// TIA Portal V18 export
// export: Created 2026-06-11T19:03:46.1512647Z, ExportSetting WithDefaults, DisplayName Totally Integrated Automation Portal, DisplayVersion V18, DisplayName TIA Portal Openness, DisplayVersion V18, DisplayName TIA Portal Version Control Interface, DisplayVersion V18, DisplayName STEP 7 Professional, DisplayVersion V18, DisplayName STEP 7 Safety, DisplayVersion V18, DisplayName WinCC Professional, DisplayVersion V18
Screen "scadabai5"  1920x1080, Number=6
  ScreenLayer 
    GraphicView "Graphic view_1" at 0,0 size 1920x1080  Picture=anh nen
    Circle "Circle_1" at 8,51 size 19x19
    Circle "Circle_2" at 8,68 size 19x19
    Circle "Circle_3" at 8,87 size 19x19
    Circle "Circle_4" at 180,52 size 19x19
    Circle "Circle_5" at 181,70 size 19x19
    Circle "Circle_6" at 250,175 size 19x19
    Circle "Circle_7" at 122,242 size 18x18
    Circle "Circle_8" at 122,259 size 18x18
    Circle "Circle_9" at 122,277 size 19x19
    Circle "Circle_10" at 86,316 size 19x19
    Circle "Circle_11" at 188,316 size 19x19
    Circle "Circle_12" at 283,316 size 19x19
    GraphicView "Graphic view_2" at 194,49 size 90x150  Picture=bon
    Circle "Circle_13" at 217,166 size 32x32
    Circle "Circle_14" at 39,392 size 19x19
    Circle "Circle_15" at 144,392 size 17x17
    Circle "Circle_16" at 238,391 size 17x17
    Button "Button_5" at 1704,197 size 39x37  Mode=Text, TextOn="Text"
    Button "Button_6" at 1740,45 size 171x35  Mode=Text, TextOff="TRANSPORT GROUP", TextOn="Text"
    Button "Button_7" at 1742,85 size 171x35  Mode=Text, TextOff="GAS FLOW GROUP", TextOn="Text"
    Button "Button_8" at 1741,116 size 172x37  Mode=Text, TextOff="LUB GROUP", TextOn="Text"
    Button "Button_9" at 1742,154 size 170x36  Mode=Text, TextOff="CEMENT MILL GROUP", TextOn="Text"
    Button "Button_10" at 1742,198 size 171x35  Mode=Text, TextOff="CM FEED GROUP", TextOn="Text"
    Button "Button_11" at 1698,242 size 220x24  Mode=Text, TextOff="ALARM RESET", TextOn="Text"
    Button "Button_12" at 1698,268 size 220x22  Mode=Text, TextOff="CM DAMFERS", TextOn="Text"
    Button "Button_13" at 1698,293 size 220x34  Mode=Text, TextOff="INTERLOCKS", TextOn="Text"
    TextField "Text field_1" at 228,171 size 12x19  Text="M"
    Circle "Circle_17" at 86,152 size 30x30
    Circle "Circle_18" at 118,152 size 30x30
    Circle "Circle_19" at 73,77 size 33x33
    TextField "Text field_2" at 95,158 size 12x19  Text="M"
    TextField "Text field_3" at 129,157 size 12x19  Text="M"
    TextField "Text field_4" at 83,83 size 12x19  Text="M"
    Circle "Circle_20" at 257,257 size 30x30
    TextField "Text field_5" at 267,264 size 12x19  Text="M"
    IOField "I/O field_1" at 53,455 size 57x22  DataFormat=Decimal, FormatPattern=99.9, Mode=InOutput
      ProcessValue := AI_B5_CA_Fan_Motor_DE_Temp
    IOField "I/O field_2" at 54,485 size 54x22  DataFormat=Decimal, FormatPattern=99.9, Mode=InOutput
      ProcessValue := AI_B5_CA_Fan_Motor_NDE_Temp
    IOField "I/O field_3" at 54,515 size 55x22  DataFormat=Decimal, FormatPattern=99.9, Mode=InOutput
      ProcessValue := AI_B5_CA_Fan_DE_Temp
    IOField "I/O field_4" at 157,455 size 55x22  DataFormat=Decimal, FormatPattern=99.9, Mode=InOutput
      ProcessValue := AI_B5_CA_Fan_NDE_Temp
    IOField "I/O field_5" at 156,488 size 56x22  DataFormat=Decimal, FormatPattern=99.9, Mode=InOutput
      ProcessValue := AI_B5_CA_Fan_DE_Vib
    IOField "I/O field_6" at 155,516 size 58x24  DataFormat=Decimal, FormatPattern=99.9, Mode=InOutput
      ProcessValue := AI_B5_CA_Fan_NDE_Vib
    IOField "I/O field_7" at 259,453 size 53x24  DataFormat=Decimal, FormatPattern=999.9, Mode=InOutput
      ProcessValue := AI_B5_SP_700FN03
    IOField "I/O field_8" at 259,483 size 54x22  DataFormat=Decimal, FormatPattern=999.9, Mode=InOutput
      ProcessValue := AI_B5_SP_700HES01
    IOField "I/O field_9" at 259,512 size 54x23  DataFormat=Decimal, FormatPattern=99.9, Mode=InOutput
      ProcessValue := AI_B5_SP_700DA4
    IOField "I/O field_10" at 482,376 size 59x17  DataFormat=Decimal, FormatPattern=99.9, Mode=InOutput
      ProcessValue := AI_B5_SP_700DA6
    IOField "I/O field_11" at 482,396 size 59x17  DataFormat=Decimal, FormatPattern=99.9, Mode=InOutput
      ProcessValue := AI_B5_SP_700DA7
    IOField "I/O field_12" at 482,416 size 59x18  DataFormat=Decimal, FormatPattern=99.9, Mode=InOutput
      ProcessValue := AI_B5_SP_700FN2_DA1
    IOField "I/O field_13" at 481,435 size 59x17  DataFormat=Decimal, FormatPattern=99.9, Mode=InOutput
      ProcessValue := AI_B5_Sep_Motor_Top_Temp
    IOField "I/O field_14" at 481,455 size 59x17  DataFormat=Decimal, FormatPattern=99.9, Mode=InOutput
      ProcessValue := AI_B5_Sep_Bottom_Bear_Temp
    IOField "I/O field_15" at 481,476 size 59x17  DataFormat=Decimal, FormatPattern=999.9, Mode=InOutput
      ProcessValue := AI_B5_Trend_Val_1
    IOField "I/O field_16" at 482,513 size 57x17  DataFormat=Decimal, FormatPattern=999.9, Mode=InOutput
      ProcessValue := AI_B5_Trend_Val_2
    IOField "I/O field_17" at 482,536 size 58x18  DataFormat=Decimal, FormatPattern=999.9, Mode=InOutput
      ProcessValue := AI_B5_Trend_Val_3
    IOField "I/O field_18" at 647,377 size 59x17  DataFormat=Decimal, FormatPattern=999.9, Mode=InOutput
      ProcessValue := AI_B5_700FN03_RPM
    IOField "I/O field_19" at 646,397 size 59x18  DataFormat=Decimal, FormatPattern=999.9, Mode=InOutput
      ProcessValue := AI_B5_700HES01_Flow
    IOField "I/O field_20" at 647,414 size 59x17  DataFormat=Decimal, FormatPattern=99.9, Mode=InOutput
      ProcessValue := AI_B5_700FN10_Speed
    IOField "I/O field_21" at 647,436 size 59x17  DataFormat=Decimal, FormatPattern=999.9, Mode=InOutput
      ProcessValue := AI_B5_700CM01_Current
    IOField "I/O field_22" at 647,457 size 59x17  DataFormat=Decimal, FormatPattern=999.9, Mode=InOutput
      ProcessValue := AI_B5_Lub_Stop_Time
    IOField "I/O field_23" at 647,479 size 58x17  DataFormat=Decimal, FormatPattern=999.9, Mode=InOutput
      ProcessValue := AI_B5_Main_Drive_ReHealth
    IOField "I/O field_24" at 334,648 size 58x23  DataFormat=Decimal, FormatPattern=99.9, Mode=InOutput
      ProcessValue := AI_B5_CM_LRS_IN
    IOField "I/O field_25" at 334,674 size 58x22  DataFormat=Decimal, FormatPattern=99.9, Mode=InOutput
      ProcessValue := AI_B5_CM_LRS_OUT
    IOField "I/O field_26" at 156,583 size 54x23  DataFormat=Decimal, FormatPattern=99.9, Mode=InOutput
      ProcessValue := AI_B5_CM_Mill_Oil_Temp
    IOField "I/O field_27" at 252,584 size 53x22  DataFormat=Decimal, FormatPattern=99.9, Mode=InOutput
      ProcessValue := AI_B5_CM_OilTrun_BER_Temp
    IOField "I/O field_28" at 765,382 size 59x22  DataFormat=Decimal, FormatPattern=99.9, Mode=InOutput
      ProcessValue := AI_B5_CM_OilTrun_BER2_Temp
    IOField "I/O field_29" at 876,299 size 57x26  DataFormat=Decimal, FormatPattern=99.9, Mode=InOutput
      ProcessValue := AI_B5_CM_OilPinion_BER_Temp
    IOField "I/O field_30" at 925,369 size 57x24  DataFormat=Decimal, FormatPattern=99.9, Mode=InOutput
      ProcessValue := AI_B5_CM_GB_IL_Shaft_BER
    IOField "I/O field_31" at 924,400 size 59x22  DataFormat=Decimal, FormatPattern=999.9, Mode=InOutput
      ProcessValue := AI_B5_CM_Running_Hours
    IOField "I/O field_32" at 824,88 size 59x23  DataFormat=Decimal, FormatPattern=99.9, Mode=InOutput
      ProcessValue := AI_B5_CM_PS1_1_KG
    IOField "I/O field_33" at 1062,42 size 56x23  DataFormat=Decimal, FormatPattern=99.9, Mode=InOutput
      ProcessValue := AI_B5_CM_PS1_2_KG
    IOField "I/O field_34" at 1375,249 size 56x21  DataFormat=Decimal, FormatPattern=999.9, Mode=InOutput
      ProcessValue := AI_B5_NIBS_Value
    IOField "I/O field_40" at 500,885 size 55x18  DataFormat=Decimal, FormatPattern=999.9, Mode=InOutput
      ProcessValue := AI_B5_800YF2_Flow
    IOField "I/O field_41" at 501,904 size 52x16  DataFormat=Decimal, FormatPattern=999.9, Mode=InOutput
      ProcessValue := AI_B5_Silo1_Level_Bar1
    IOField "I/O field_42" at 626,631 size 58x22  DataFormat=Decimal, FormatPattern=999.9, Mode=InOutput
      ProcessValue := AI_B5_Silo1_Level_Bar2
    IOField "I/O field_43" at 641,714 size 58x22  DataFormat=Decimal, FormatPattern=999.9, Mode=InOutput
      ProcessValue := AI_B5_Silo2_Level_Bar1
    IOField "I/O field_44" at 690,812 size 59x22  DataFormat=Decimal, FormatPattern=999.9, Mode=InOutput
      ProcessValue := AI_B5_Silo2_Level_Bar2
    IOField "I/O field_45" at 757,909 size 58x22  DataFormat=Decimal, FormatPattern=99.9, Mode=InOutput
      ProcessValue := AI_B5_700FN01_Speed
    IOField "I/O field_46" at 878,891 size 52x22  DataFormat=Decimal, FormatPattern=99.9, Mode=InOutput
      ProcessValue := AI_B5_700FN02_Speed
    IOField "I/O field_47" at 954,696 size 58x22  DataFormat=Decimal, FormatPattern=99.9, Mode=InOutput
      ProcessValue := AI_B5_700AS07_Speed
    IOField "I/O field_48" at 1062,835 size 51x22  DataFormat=Decimal, FormatPattern=999.9, Mode=InOutput
      ProcessValue := AI_B5_700AS08_Flow
    IOField "I/O field_49" at 1137,789 size 58x22  DataFormat=Decimal, FormatPattern=99.9, Mode=InOutput
      ProcessValue := AI_B5_700FN09_Speed
    IOField "I/O field_50" at 1131,949 size 58x22  DataFormat=Decimal, FormatPattern=99.9, Mode=InOutput
      ProcessValue := AI_B5_700SFM01_Speed
    IOField "I/O field_51" at 1381,929 size 58x21  DataFormat=Decimal, FormatPattern=999.9, Mode=InOutput
      ProcessValue := AI_B5_700DA1_Flow
    IOField "I/O field_52" at 1391,790 size 58x21  DataFormat=Decimal, FormatPattern=999.9, Mode=InOutput
      ProcessValue := AI_B5_700DA4_Flow
    IOField "I/O field_53" at 1768,859 size 58x24  DataFormat=Decimal, FormatPattern=99.9, Mode=InOutput
      ProcessValue := AI_B5_700DA6_Temp
    IOField "I/O field_54" at 465,956 size 49x16  DataFormat=Decimal, FormatPattern=99.9, Mode=InOutput
      ProcessValue := AI_B5_700DA7_Temp
    IOField "I/O field_55" at 523,957 size 49x16  DataFormat=Decimal, FormatPattern=999.9, Mode=InOutput
      ProcessValue := AI_B5_700BL1_Load
    IOField "I/O field_56" at 246,862 size 58x23  DataFormat=Decimal, FormatPattern=999.9, Mode=InOutput
      ProcessValue := AI_B5_700BL2_Load
    Circle "Circle_21" at 286,82 size 32x32
    TextField "Text field_6" at 296,88 size 12x19  Text="M"
    Circle "Circle_22" at 86,416 size 30x30
    Circle "Circle_23" at 192,416 size 28x28
    Circle "Circle_24" at 288,414 size 31x31
    Circle "Circle_25" at 98,612 size 18x18
    Circle "Circle_26" at 162,612 size 18x18
    Circle "Circle_27" at 226,613 size 18x18
    Circle "Circle_28" at 74,705 size 25x25
    TextField "Text field_7" at 94,423 size 12x19  Text="M"
    TextField "Text field_8" at 201,421 size 12x19  Text="M"
    TextField "Text field_9" at 299,421 size 12x19  Text="M"
    TextField "Text field_10" at 81,708 size 12x19  Text="M"
    Circle "Circle_29" at 138,706 size 25x25
    Circle "Circle_30" at 177,706 size 25x25
    Circle "Circle_31" at 177,772 size 25x25
    Circle "Circle_32" at 138,772 size 25x25
    Circle "Circle_33" at 73,772 size 25x25
    TextField "Text field_11" at 144,709 size 12x19  Text="M"
    TextField "Text field_12" at 184,709 size 12x19  Text="M"
    TextField "Text field_13" at 184,774 size 12x19  Text="M"
    TextField "Text field_14" at 145,775 size 12x19  Text="M"
    TextField "Text field_15" at 80,776 size 12x19  Text="M"
    Circle "Circle_34" at 74,846 size 25x25
    Circle "Circle_35" at 138,845 size 25x25
    Circle "Circle_36" at 73,916 size 25x25
    Circle "Circle_37" at 142,916 size 17x17
    Circle "Circle_38" at 176,915 size 17x17
    Circle "Circle_39" at 210,915 size 17x17
    Circle "Circle_40" at 243,916 size 17x17
    Circle "Circle_41" at 141,950 size 17x17
    TextField "Text field_16" at 81,848 size 12x19  Text="M"
    TextField "Text field_17" at 144,848 size 12x19  Text="M"
    Circle "Circle_42" at 408,727 size 17x17
    Circle "Circle_43" at 407,746 size 17x17
    Circle "Circle_44" at 408,764 size 17x17
    Bar "Bar_1" at 1622,837 size 85x126  CountSubDivisions=2, IntegerDigits=2, LargeTickLabelingStep=1, MaximumValue=25, Precision=2
    Bar "Bar_2" at 1914,794 size 86x124  CountSubDivisions=2, IntegerDigits=2, LargeTickLabelingStep=1, MaximumValue=25, Precision=2
    IOField "I/O field_57" at 945,188 size 59x21  DataFormat=Decimal, FormatPattern=999.9, Mode=InOutput
      ProcessValue := AI_B5_700AS9_Flow
    IOField "I/O field_58" at 946,213 size 58x23  DataFormat=Decimal, FormatPattern=99.9, Mode=InOutput
      ProcessValue := AI_B5_700FN13_Speed
    Button "Button_14" at 98,190 size 39x23  Mode=Text, TextOff="Text", TextOn="Text"
    Button "Button_15" at 18,454 size 33x24  Mode=Text, TextOff="Text", TextOn="Text"
    Button "Button_16" at 18,485 size 33x24  Mode=Text, TextOff="Text", TextOn="Text"
    Button "Button_17" at 119,454 size 34x23  Mode=Text, TextOff="Text", TextOn="Text"
    Button "Button_18" at 119,486 size 33x23  Mode=Text, TextOff="Text", TextOn="Text"
    Button "Button_19" at 223,486 size 33x23  Mode=Text, TextOff="Text", TextOn="Text"
    Button "Button_20" at 223,455 size 33x23  Mode=Text, TextOff="Text", TextOn="Text"
    Button "Button_21" at 249,950 size 66x33  Mode=Text, TextOff="LOS", TextOn="Text"
    Button "Button_22" at 11,711 size 60x49  Mode=Text, TextOff="LQ 61", TextOn="Text"
    Button "Button_23" at 13,775 size 58x46  Mode=Text, TextOff="LQ 62", TextOn="Text"
    Button "Button_24" at 13,836 size 57x49  Mode=Text, TextOff="ELS", TextOn="Text"
    Button "Button_25" at 13,922 size 58x55  Mode=Text, TextOff="LQ 63", TextOn="Text"
    Circle "Circle_45" at 560,578 size 33x33
    TextField "Text field_18" at 570,585 size 12x19  Text="M"
    Circle "Circle_46" at 796,584 size 32x32
    Circle "Circle_47" at 868,585 size 29x29
    TextField "Text field_19" at 805,589 size 12x19  Text="M"
    TextField "Text field_20" at 878,590 size 12x19  Text="M"
    Circle "Circle_48" at 772,764 size 33x33
    TextField "Text field_21" at 784,772 size 12x19  Text="M"
    Circle "Circle_49" at 769,860 size 33x33
    TextField "Text field_22" at 779,867 size 12x19  Text="M"
    Circle "Circle_50" at 740,855 size 22x22
    TextField "Text field_23" at 745,856 size 12x19  Text="M"
    Circle "Circle_51" at 898,860 size 22x22
    TextField "Text field_24" at 903,861 size 12x19  Text="M"
    Circle "Circle_52" at 895,947 size 14x14
    Circle "Circle_53" at 895,961 size 14x14
    Circle "Circle_54" at 970,921 size 31x31
    TextField "Text field_25" at 980,926 size 12x19  Text="M"
    Circle "Circle_55" at 1014,921 size 31x31
    TextField "Text field_26" at 1024,928 size 12x19  Text="M"
    Circle "Circle_56" at 808,464 size 19x19
    Circle "Circle_57" at 833,460 size 25x25
    Circle "Circle_58" at 877,461 size 25x25
    Circle "Circle_59" at 908,464 size 19x19
    Circle "Circle_60" at 985,464 size 19x19
    Circle "Circle_61" at 1009,458 size 25x25
    Circle "Circle_62" at 1289,433 size 33x33
    Circle "Circle_63" at 1086,464 size 19x19
    TextField "Text field_27" at 839,464 size 12x19  Text="M"
    TextField "Text field_28" at 883,464 size 12x19  Text="M"
    TextField "Text field_30" at 1299,440 size 12x19  Text="M"
    Circle "Circle_64" at 934,314 size 41x41
    TextField "Text field_31" at 948,326 size 12x19  Text="M"
    Circle "Circle_65" at 958,115 size 33x33
    TextField "Text field_32" at 968,120 size 12x19  Text="M"
    Circle "Circle_66" at 1100,209 size 30x30
    TextField "Text field_33" at 1110,213 size 12x19  Text="M"
    Circle "Circle_67" at 1147,62 size 33x33
    TextField "Text field_34" at 1156,68 size 12x19  Text="M"
    Circle "Circle_68" at 1188,95 size 18x18
    Circle "Circle_69" at 1316,52 size 19x19
    Circle "Circle_70" at 1317,70 size 19x19
    Circle "Circle_71" at 1335,166 size 19x19
    Circle "Circle_72" at 1357,79 size 31x31
    Circle "Circle_73" at 1357,157 size 30x30
    Circle "Circle_74" at 1459,135 size 30x30
    Circle "Circle_75" at 1454,218 size 30x30
    Circle "Circle_76" at 1298,282 size 30x30
    TextField "Text field_35" at 1308,287 size 12x19  Text="M"
    TextField "Text field_36" at 1368,85 size 12x19  Text="M"
    TextField "Text field_37" at 1430,152 size 12x19  Text="M"
    TextField "Text field_38" at 1367,164 size 12x19  Text="M"
    TextField "Text field_39" at 1463,224 size 12x19  Text="M"
    Circle "Circle_77" at 1155,920 size 22x22
    Circle "Circle_78" at 1236,385 size 19x19
    Circle "Circle_79" at 1236,406 size 19x19
    Circle "Circle_80" at 1379,495 size 19x19
    Circle "Circle_81" at 1489,372 size 19x19
    Circle "Circle_82" at 1489,391 size 19x19
    Circle "Circle_83" at 1272,530 size 19x19
    Circle "Circle_84" at 1401,488 size 36x36
    TextField "Text field_40" at 1413,496 size 12x19  Text="M"
    Circle "Circle_85" at 1526,479 size 36x36
    TextField "Text field_41" at 1536,488 size 12x19  Text="M"
    Circle "Circle_86" at 1603,397 size 31x31
    TextField "Text field_42" at 1614,404 size 12x19  Text="M"
    Circle "Circle_87" at 1532,399 size 31x31
    TextField "Text field_43" at 1542,405 size 12x19  Text="M"
    Circle "Circle_88" at 1713,481 size 31x31
    TextField "Text field_44" at 1722,488 size 12x19  Text="M"
    Circle "Circle_89" at 1564,490 size 19x19
    Circle "Circle_90" at 1672,373 size 19x19
    Circle "Circle_91" at 1673,393 size 19x19
    Circle "Circle_92" at 1693,488 size 19x19
    Circle "Circle_93" at 1788,399 size 31x31
    Circle "Circle_94" at 1792,458 size 31x31
    Circle "Circle_95" at 1712,394 size 31x31
    TextField "Text field_45" at 1797,406 size 12x19  Text="M"
    TextField "Text field_46" at 1722,400 size 12x19  Text="M"
    TextField "Text field_47" at 1801,465 size 12x19  Text="M"
    Circle "Circle_96" at 1580,600 size 31x31
    TextField "Text field_48" at 1590,608 size 12x19  Text="M"
    Circle "Circle_97" at 1473,769 size 31x31
    TextField "Text field_49" at 1483,774 size 12x19  Text="M"
    Circle "Circle_98" at 1301,889 size 31x31
    TextField "Text field_50" at 1311,894 size 12x19  Text="M"
    Circle "Circle_99" at 1234,888 size 31x31
    TextField "Text field_51" at 1244,894 size 12x19  Text="M"
    Circle "Circle_100" at 1411,885 size 17x17
    Circle "Circle_101" at 1687,769 size 31x31
    TextField "Text field_52" at 1696,774 size 12x19  Text="M"
    Button "Button_26" at 1529,929 size 78x23  Mode=Text, TextOff="SELECTED", TextOn="Text"
    Circle "Circle_102" at 1506,840 size 20x20
    Circle "Circle_103" at 1723,842 size 20x20
    Button "Button_28" at 179,1024 size 173x20  Mode=Text, TextOff="REPORT", TextOn="Text"
    Button "Button_29" at 178,1049 size 172x24  Mode=Text, TextOff="TRENDS", TextOn="Text"
    Button "Button_30" at 357,1024 size 167x20  Mode=Text, TextOff="RAW MILL", TextOn="Text"
    Button "Button_31" at 355,1048 size 168x25  Mode=Text, TextOff="ALARM", TextOn="Text"
    Button "Button_32" at 527,1021 size 171x23  Mode=Text, TextOff="BLENDING SILO", TextOn="Text"
    Button "Button_33" at 527,1049 size 172x23  Mode=Text, TextOff="FLYASH SILO", TextOn="Text"
    Button "Button_34" at 700,1021 size 172x25  Mode=Text, TextOff="COAL MILL", TextOn="Text"
    Button "Button_35" at 700,1047 size 173x25  Mode=Text, TextOff="INSTRUCTIONS", TextOn="Text"
    Button "Button_36" at 875,1021 size 169x25  Mode=Text, TextOff="GREATE COOLER", TextOn="Text"
    Button "Button_37" at 1047,1018 size 171x25  Mode=Text, TextOff="KILN GROUP", TextOn="Text"
    Button "Button_38" at 1220,1020 size 175x25  Mode=Text, TextOff="HOPPER FEEDING", TextOn="Text"
    Button "Button_39" at 1398,1018 size 169x25  Mode=Text, TextOff="CEM MILL GROUP", TextOn="Text"
    Button "Button_40" at 1566,1019 size 180x25  Mode=Text, TextOff="EXTR.& PACKING", TextOn="Text"
    Button "Button_41" at 874,1047 size 172x25  Mode=Text, TextOff="RUNNING HOURS", TextOn="Text"
    Button "Button_42" at 1047,1047 size 171x25  Mode=Text, TextOff="SPARE", TextOn="Text"
    Button "Button_43" at 1222,1047 size 170x25  Mode=Text, TextOff="HOOTER", TextOn="Text"
    Button "Button_44" at 1396,1048 size 169x25  Mode=Text, TextOff="EXIT", TextOn="Text"
    Button "Button_45" at 1565,1048 size 180x25  Mode=Text, TextOff="ABOUT", TextOn="Text"
    IOField "I/O field_35" at 500,865 size 55x18  DataFormat=Decimal, FormatPattern=99.9, Mode=InOutput
      ProcessValue := AI_B5_800DC1_Temp
    IOField "I/O field_36" at 500,845 size 55x18  DataFormat=Decimal, FormatPattern=99.9, Mode=InOutput
      ProcessValue := AI_B5_800DC2_Temp
    Bar "Bar_3" at 1822,834 size 85x126  CountSubDivisions=2, IntegerDigits=2, LargeTickLabelingStep=1, MaximumValue=25, Precision=2
    IOField "I/O field_37" at 500,825 size 55x18  DataFormat=Decimal, FormatPattern=99.9, Mode=InOutput
      ProcessValue := AI_B5_800FN1_Speed
    IOField "I/O field_38" at 500,805 size 55x18  DataFormat=Decimal, FormatPattern=99.9, Mode=InOutput
      ProcessValue := AI_B5_800FN2_Speed
    IOField "I/O field_39" at 500,785 size 55x18  DataFormat=Decimal, FormatPattern=999.9, Mode=InOutput
      ProcessValue := AI_B5_800YF1_Flow
    Button "Button_27" at 1756,929 size 78x23  Mode=Text, TextOff="SELECTED", TextOn="Text"
    Button "Button_1" at 1704,159 size 39x37  Mode=Text, TextOn="Text"
    Button "Button_2" at 1704,121 size 39x37  Mode=Text, TextOn="Text"
    Button "Button_3" at 1704,83 size 39x37  Mode=Text, TextOn="Text"
    Button "Button_4" at 1704,45 size 39x37  Mode=Text, TextOn="Text"
    Circle "Circle_104" at 1292,522 size 33x33
    TextField "Text field_29" at 1304,530 size 12x19  Text="M"
    Circle "Circle_105" at 1055,460 size 24x24
    TextField "Text field_53" at 1061,463 size 12x19  Text="M"
    TextField "Text field_54" at 1015,462 size 12x19  Text="M"
    Circle "Circle_106" at 1082,587 size 29x29
    TextField "Text field_55" at 1090,594 size 12x19  Text="M"
    Button "Btn_Enter_System_4" at 1806,0 size 114x38  Mode=Text, StyleItem=Button, TextOff="Mh login", TextOn="Text"
      VisibilityAnimation "VisibilityAnimation"  RangeEnd=99, RangeStart=1
        tag Logged_In
      on Click: ActivateScreen(Screen name := Login/out, Object number := 0)
    TextField "Text_field_Unit_I/O field_1" at 118,455 size 50x22  Text="<body><p>°C</p></body>"
    TextField "Text_field_Unit_I/O field_2" at 116,485 size 50x22  Text="<body><p>°C</p></body>"
    TextField "Text_field_Unit_I/O field_3" at 117,515 size 50x22  Text="<body><p>°C</p></body>"
    TextField "Text_field_Unit_I/O field_4" at 220,455 size 50x22  Text="<body><p>°C</p></body>"
    TextField "Text_field_Unit_I/O field_5" at 220,488 size 50x22  Text="<body><p>mm/s</p></body>"
    TextField "Text_field_Unit_I/O field_6" at 221,516 size 50x24  Text="<body><p>mm/s</p></body>"
    TextField "Text_field_Unit_I/O field_7" at 320,453 size 50x24  Text="<body><p>L/h</p></body>"
    TextField "Text_field_Unit_I/O field_8" at 321,483 size 50x22  Text="<body><p>L/h</p></body>"
    TextField "Text_field_Unit_I/O field_9" at 321,512 size 50x23  Text="<body><p>Hz</p></body>"
    TextField "Text_field_Unit_I/O field_10" at 549,376 size 50x17  Text="<body><p>Hz</p></body>"
    TextField "Text_field_Unit_I/O field_11" at 549,396 size 50x17  Text="<body><p>Hz</p></body>"
    TextField "Text_field_Unit_I/O field_12" at 549,416 size 50x18  Text="<body><p>Hz</p></body>"
    TextField "Text_field_Unit_I/O field_13" at 548,435 size 50x17  Text="<body><p>°C</p></body>"
    TextField "Text_field_Unit_I/O field_14" at 548,455 size 50x17  Text="<body><p>°C</p></body>"
    TextField "Text_field_Unit_I/O field_15" at 548,476 size 50x17  Text="<body><p>%</p></body>"
    TextField "Text_field_Unit_I/O field_16" at 547,513 size 50x17  Text="<body><p>%</p></body>"
    TextField "Text_field_Unit_I/O field_17" at 548,536 size 50x18  Text="<body><p>%</p></body>"
    TextField "Text_field_Unit_I/O field_18" at 714,377 size 50x17  Text="<body><p>RPM</p></body>"
    TextField "Text_field_Unit_I/O field_19" at 713,397 size 50x18  Text="<body><p>L/h</p></body>"
    TextField "Text_field_Unit_I/O field_20" at 714,414 size 50x17  Text="<body><p>Hz</p></body>"
    TextField "Text_field_Unit_I/O field_21" at 714,436 size 50x17  Text="<body><p>A</p></body>"
    TextField "Text_field_Unit_I/O field_22" at 714,457 size 50x17  Text="<body><p>Sec</p></body>"
    TextField "Text_field_Unit_I/O field_23" at 713,479 size 50x17  Text="<body><p>Sec</p></body>"
    TextField "Text_field_Unit_I/O field_24" at 400,648 size 50x23  Text="<body><p>°C</p></body>"
    TextField "Text_field_Unit_I/O field_25" at 400,674 size 50x22  Text="<body><p>°C</p></body>"
    TextField "Text_field_Unit_I/O field_26" at 218,583 size 50x23  Text="<body><p>°C</p></body>"
    TextField "Text_field_Unit_I/O field_27" at 313,584 size 50x22  Text="<body><p>°C</p></body>"
    TextField "Text_field_Unit_I/O field_28" at 832,382 size 50x22  Text="<body><p>°C</p></body>"
    TextField "Text_field_Unit_I/O field_29" at 941,299 size 50x26  Text="<body><p>°C</p></body>"
    TextField "Text_field_Unit_I/O field_30" at 990,369 size 50x24  Text="<body><p>°C</p></body>"
    TextField "Text_field_Unit_I/O field_31" at 991,400 size 50x22  Text="<body><p>Hr</p></body>"
    TextField "Text_field_Unit_I/O field_32" at 891,88 size 50x23  Text="<body><p>bar</p></body>"
    TextField "Text_field_Unit_I/O field_33" at 1126,42 size 50x23  Text="<body><p>bar</p></body>"
    TextField "Text_field_Unit_I/O field_34" at 1439,249 size 50x21  Text="<body><p>A</p></body>"
    TextField "Text_field_Unit_I/O field_40" at 563,885 size 50x18  Text="<body><p>L/h</p></body>"
    TextField "Text_field_Unit_I/O field_41" at 561,904 size 50x16  Text="<body><p>%</p></body>"
    TextField "Text_field_Unit_I/O field_42" at 692,631 size 50x22  Text="<body><p>%</p></body>"
    TextField "Text_field_Unit_I/O field_43" at 707,714 size 50x22  Text="<body><p>%</p></body>"
    TextField "Text_field_Unit_I/O field_44" at 757,812 size 50x22  Text="<body><p>%</p></body>"
    TextField "Text_field_Unit_I/O field_45" at 823,909 size 50x22  Text="<body><p>Hz</p></body>"
    TextField "Text_field_Unit_I/O field_46" at 938,891 size 50x22  Text="<body><p>Hz</p></body>"
    TextField "Text_field_Unit_I/O field_47" at 1020,696 size 50x22  Text="<body><p>Hz</p></body>"
    TextField "Text_field_Unit_I/O field_48" at 1121,835 size 50x22  Text="<body><p>L/h</p></body>"
    TextField "Text_field_Unit_I/O field_49" at 1203,789 size 50x22  Text="<body><p>Hz</p></body>"
    TextField "Text_field_Unit_I/O field_50" at 1197,949 size 50x22  Text="<body><p>Hz</p></body>"
    TextField "Text_field_Unit_I/O field_51" at 1447,929 size 50x21  Text="<body><p>L/h</p></body>"
    TextField "Text_field_Unit_I/O field_52" at 1457,790 size 50x21  Text="<body><p>L/h</p></body>"
    TextField "Text_field_Unit_I/O field_53" at 1834,859 size 50x24  Text="<body><p>°C</p></body>"
    TextField "Text_field_Unit_I/O field_54" at 522,956 size 50x16  Text="<body><p>°C</p></body>"
    TextField "Text_field_Unit_I/O field_55" at 580,957 size 50x16  Text="<body><p>A</p></body>"
    TextField "Text_field_Unit_I/O field_56" at 312,862 size 50x23  Text="<body><p>A</p></body>"
    TextField "Text_field_Unit_I/O field_57" at 1012,188 size 50x21  Text="<body><p>L/h</p></body>"
    TextField "Text_field_Unit_I/O field_58" at 1012,213 size 50x23  Text="<body><p>Hz</p></body>"
    TextField "Text_field_Unit_I/O field_35" at 563,865 size 50x18  Text="<body><p>°C</p></body>"
    TextField "Text_field_Unit_I/O field_36" at 563,845 size 50x18  Text="<body><p>°C</p></body>"
    TextField "Text_field_Unit_I/O field_37" at 563,825 size 50x18  Text="<body><p>Hz</p></body>"
    TextField "Text_field_Unit_I/O field_38" at 563,805 size 50x18  Text="<body><p>Hz</p></body>"
    TextField "Text_field_Unit_I/O field_39" at 563,785 size 50x18  Text="<body><p>L/h</p></body>"
